FUNCTION_BLOCK FB_SolenoidPair
VAR_INPUT
END_VAR
VAR_OUTPUT
END_VAR
VAR_IN_OUT
END_VAR
VAR
    {attribute 'pytmc' := '
        pv: Valve:01:Open
        io: io
        field: ZNAM "CLOSE"
        field: ONAM "OPEN"
     '}
    q_xDO1 AT %Q*	:	BOOL;
    {attribute 'pytmc' := '
        pv: Valve:02:Open
        io: io
        field: ZNAM "CLOSE"
        field: ONAM "OPEN"
     '}
    q_xDO2 AT %Q*	:	BOOL;

    {attribute 'pytmc' := '
        pv: Switch
        io: o
     '}
    i_xEpics AT %I* : BOOL; // open A when False, open B when True

    {attribute 'pytmc' := '
        pv: Debug
        io: o
     '}
    i_xDebug AT %I* : BOOL; // if True, do not set valves according to i_xEpics
END_VAR

(* If debug, set independently. Else, only open one valve according to i_xEpics *)
IF NOT i_xDebug THEN
    q_xDO1 := NOT i_xEpics;
    q_xDO2 := i_xEpics;
END_IF

END_FUNCTION_BLOCK

(* stored: Version 1.1.0.1, ProductVersion 3.1.4024.12
   POU FB_SolenoidPair: Id {23ddf2e7-415d-4237-9e6d-fcc92e4bc96b}, SpecialFunc None *)
